Staubli VAL3: Form_ScaraRobot.pgx

public program Form_ScaraRobot()
begin
  //为Scara机器人主界面
  //选择示教产品的类型


 call Form_PattenS("Scara1.0:主界面","示教Home,示教TCP,示教码垛,产品编辑,,选项,高级,退出","F1,F2,F3,F4,F5,F6,F7,F8")
 call Control_Scara()

end
